// TIA Portal V21 export
DATA_BLOCK "Calc"   // DB1
{ S7_Optimized_Access := 'TRUE' }
// stored: MemoryReserve 100
   VAR
      reale : Array[0..100] of LReal;
      tempociclo : LReal;
      tempociclo_T : LReal;
      interi : Array[0..10] of Int;
      tempo : LReal;
      pulse : Array[0..30] of Bool;
   END_VAR
BEGIN
END_DATA_BLOCK
